FUNCTION CheckBounds : DINT
VAR_INPUT
	index, lower, upper 	: DINT;
END_VAR
VAR
END_VAR

IF index<lower THEN
	CheckBounds_ErrCnt := CheckBounds_ErrCnt + 1;
	CheckBounds := lower;
ELSIF index>upper THEN
	CheckBounds_ErrCnt := CheckBounds_ErrCnt + 1;
	CheckBounds := upper;
ELSE
	CheckBounds := index;
END_IF

END_FUNCTION

(* stored: Version 1.1.0.1, ProductVersion 3.1.4024.9
   POU CheckBounds: Id {629469e7-baf7-4e9a-90d8-aa17884ceaa5}, SpecialFunc CheckBounds *)
